// Mitsubishi GX Works2 project: 과정 평가 문항 2   PLC: Q03UDV

PROGRAM MAIN
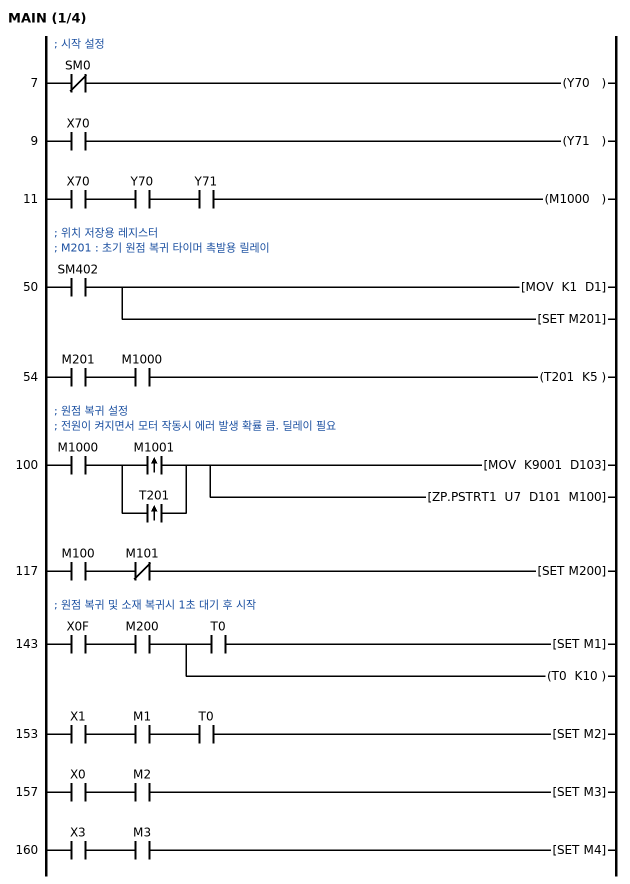
; 시작 설정
7     LDI     SM0
      OUT     Y70
9     LD      X70
      OUT     Y71
11    LD      X70
      AND     Y70
      AND     Y71
      OUT     M1000
; 위치 저장용 레지스터
; M201 : 초기 원점 복귀 타이머 촉발용 릴레이
50    LD      SM402
      MOV     K1 D1
      SET     M201
54    LD      M201
      AND     M1000
      OUT     T201 K5
; 원점 복귀 설정
; 전원이 켜지면서 모터 작동시 에러 발생 확률 큼. 딜레이 필요
100   LD      M1000
      LDP     M1001
      ORP     T201
      ANB
      MOV     K9001 D103
      ZP.PSTRT1 U7 D101 M100
117   LD      M100
      ANI     M101
      SET     M200
; 원점 복귀 및 소재 복귀시 1초 대기 후 시작
143   LD      X0F
      AND     M200
      MPS
      AND     T0
      SET     M1
      MPP
      OUT     T0 K10
153   LD      X1
      AND     M1
      AND     T0
      SET     M2
157   LD      X0
      AND     M2
      SET     M3
160   LD      X3
      AND     M3
      SET     M4
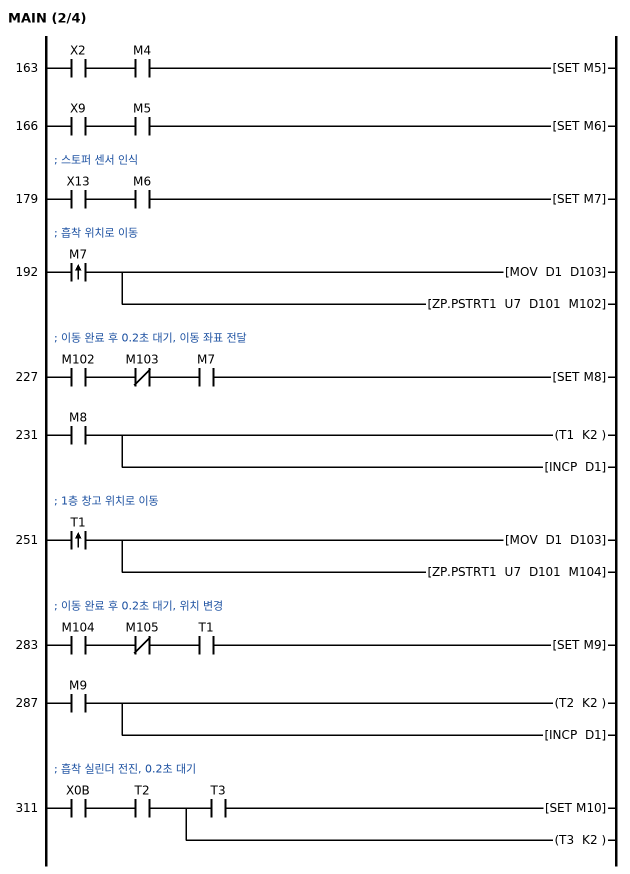
163   LD      X2
      AND     M4
      SET     M5
166   LD      X9
      AND     M5
      SET     M6
; 스토퍼 센서 인식
179   LD      X13
      AND     M6
      SET     M7
; 흡착 위치로 이동
192   LDP     M7
      MOV     D1 D103
      ZP.PSTRT1 U7 D101 M102
; 이동 완료 후 0.2초 대기, 이동 좌표 전달
227   LD      M102
      ANI     M103
      AND     M7
      SET     M8
231   LD      M8
      OUT     T1 K2
      INCP    D1
; 1층 창고 위치로 이동
251   LDP     T1
      MOV     D1 D103
      ZP.PSTRT1 U7 D101 M104
; 이동 완료 후 0.2초 대기, 위치 변경
283   LD      M104
      ANI     M105
      AND     T1
      SET     M9
287   LD      M9
      OUT     T2 K2
      INCP    D1
; 흡착 실린더 전진, 0.2초 대기
311   LD      X0B
      AND     T2
      MPS
      AND     T3
      SET     M10
      MPP
      OUT     T3 K2
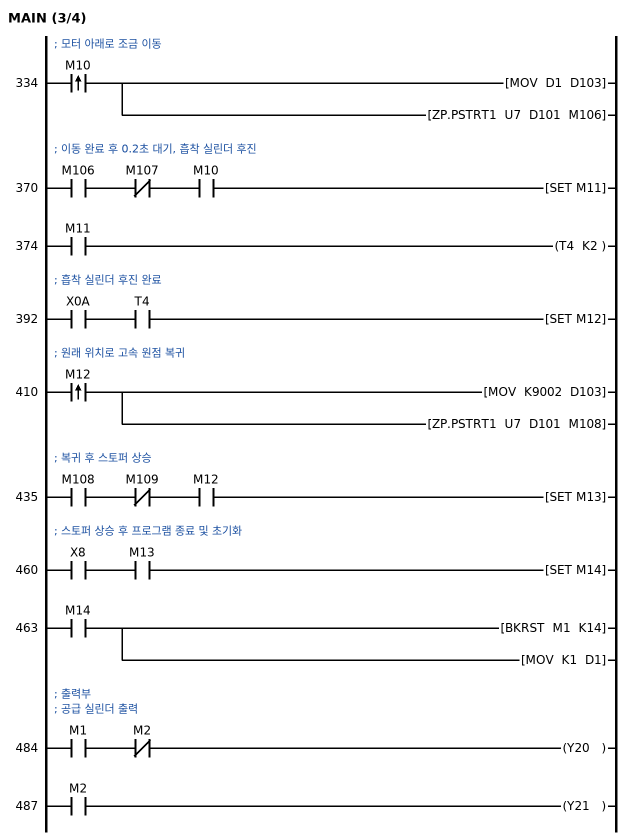
; 모터 아래로 조금 이동
334   LDP     M10
      MOV     D1 D103
      ZP.PSTRT1 U7 D101 M106
; 이동 완료 후 0.2초 대기, 흡착 실린더 후진
370   LD      M106
      ANI     M107
      AND     M10
      SET     M11
374   LD      M11
      OUT     T4 K2
; 흡착 실린더 후진 완료
392   LD      X0A
      AND     T4
      SET     M12
; 원래 위치로 고속 원점 복귀
410   LDP     M12
      MOV     K9002 D103
      ZP.PSTRT1 U7 D101 M108
; 복귀 후 스토퍼 상승
435   LD      M108
      ANI     M109
      AND     M12
      SET     M13
; 스토퍼 상승 후 프로그램 종료 및 초기화
460   LD      X8
      AND     M13
      SET     M14
463   LD      M14
      BKRST   M1 K14
      MOV     K1 D1
; 출력부
; 공급 실린더 출력
484   LD      M1
      ANI     M2
      OUT     Y20
487   LD      M2
      OUT     Y21
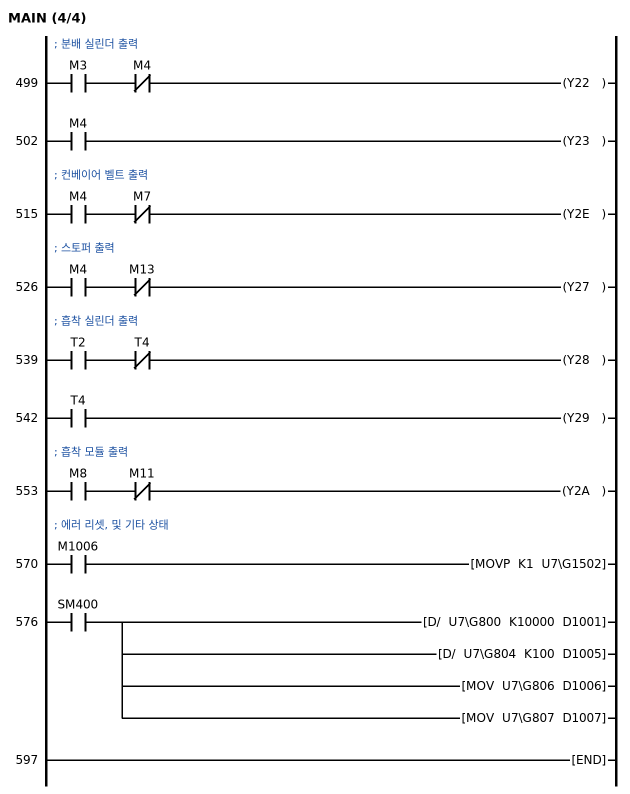
; 분배 실린더 출력
499   LD      M3
      ANI     M4
      OUT     Y22
502   LD      M4
      OUT     Y23
; 컨베이어 벨트 출력
515   LD      M4
      ANI     M7
      OUT     Y2E
; 스토퍼 출력
526   LD      M4
      ANI     M13
      OUT     Y27
; 흡착 실린더 출력
539   LD      T2
      ANI     T4
      OUT     Y28
542   LD      T4
      OUT     Y29
; 흡착 모듈 출력
553   LD      M8
      ANI     M11
      OUT     Y2A
; 에러 리셋, 및 기타 상태
570   LD      M1006
      MOVP    K1 U7\G1502
576   LD      SM400
      D/      U7\G800 K10000 D1001
      D/      U7\G804 K100 D1005
      MOV     U7\G806 D1006
      MOV     U7\G807 D1007
597   END
END_PROGRAM
